FUNCTION_BLOCK PUBLIC FB_HalfBROTAxis IMPLEMENTS I_Axis, I_Axis
VAR_INPUT
END_VAR
VAR_OUTPUT
	bCalibrated			: BOOL;		// true if absolute calibration
	bError				: BOOL;		// true if error	
END_VAR
VAR
	fbAxis				: FB_Axis2;
END_VAR

PROPERTY Busy : BOOL
GET
Busy := fbAxis.Busy;
END_GET
END_PROPERTY

{warning 'Add property implementation'}
PROPERTY Calibrated : BOOL
GET
Calibrated := bCalibrated;
END_GET
END_PROPERTY

PROPERTY Error : BOOL
GET
Error := bError;
END_GET
END_PROPERTY

END_FUNCTION_BLOCK

(* stored: Version 1.1.0.1, ProductVersion 3.1.4026.11
   POU FB_HalfBROTAxis: Id {bae85b54-65c9-4d1f-98f7-530b10d558b7}, SpecialFunc None
   Property Busy: Id {567e8af7-1006-4a9e-a236-efe3efee35b4}
   Get Get: Id {bc8cb34d-293c-40ce-ac83-5fd7efe63294}
   Property Calibrated: Id {b034059e-7dc3-4131-8628-44f1ad17bd06}
   Get Get: Id {fe3ff6d9-4050-4415-b9d6-711bddc50fae}
   Property Error: Id {e8700151-a6f7-4979-9adf-7a637755cd40}
   Get Get: Id {918a6a55-fc48-4705-8e89-8dd3c47b45de} *)
